# EPICS SNL sequencer program: HFMAGPSUSup/fsm_stage1.st
program fsm("P, RAMPTABLEDIR")

/* STAGE 1: This FSM can do basic ramping from point A to point B: no incremental ramping,
no direction work. */

/*
**************************************************************************
fsm.st

State Machine for the Hifi Cryomagnet PSU

- Reads ramp rate table from external file and stores targets/rates in
  two unsorted arrays: ramp_table_targets and their corresponding ramp_table_rates.

- The directory of the ramp file is passed to this script via the RAMPTABLEDIR
  macro. This is sourced from the st-common.cmd IOC file.

- Ramp file reading skips line 0, it is reserved for column headers.
  Subsequent file_liness have pairs of space-seperated values (target, rate)

- Ramping is incremental (ramps to interim points along the way) to avoid ramping too
  quickly if there is a comms error.

- the Direction PV sets the polarity of the ramp. When ramping from +ve to -ve
  (or vice-versa), we ramp to zero, flip the polarity, and continue the ramp to
  the user's target.

*************************************************************************
*/

/* INITIALISER VARIABLES */

double CONSTANT_INIT = 0.029;

#include "seqPVmacros.h"
%{#include <stdlib.h>}%
%{#include <stdio.h>}%
%{#include <float.h>}%

/* Turn on run-time debug messages */
option +d;

/* PV definitions */
PV(double, get_mid, "{P}:MID", Monitor);
PV(double, get_max, "{P}:MAX", Monitor);
PV(double, get_zero, "{P}:ZERO", Monitor);
PV(double, set_zero, "{P}:ZERO", Monitor);
PV(double, get_limit, "{P}:LIMIT", Monitor);
PV(string, get_pause, "{P}:PAUSE", Monitor);
PV(double, get_output, "{P}:OUTPUT", Monitor);
PV(double, get_constant, "{P}:CONSTANT", Monitor);
PV(double, get_ramp_rate, "{P}:RAMPRATE", Monitor);
PV(string, get_direction, "{P}:DIRECTION", Monitor);
PV(string, get_ramp_target, "{P}:RAMPTARGET", Monitor);
PV(string, get_output_mode, "{P}:OUTPUTMODE", Monitor);
PV(int, read_ramp_file_trigger, "{P}:READFILE", Monitor);
PV(string, get_heater_status, "{P}:HEATERSTATUS", Monitor);
PV(int, write_ramp_file_trigger, "{P}:WRITEFILE", Monitor);
PV(double, final_target, "{P}:MIDFINALTARGET", Monitor);

char ramp_table_directory[256]; assign ramp_table_directory to "{P}:RAMPTABLEDIRECTORY";
char temp_log[256];
double ramp_table_rates[64]; assign ramp_table_rates to "{P}:RAMPTABLERATES"; monitor ramp_table_rates;
double ramp_table_targets[64]; assign ramp_table_targets to "{P}:RAMPTABLETARGETS"; monitor ramp_table_targets;
int system_stable; assign system_stable to "{P}:SYSTEMSTABLE";

double ramp_time; assign ramp_time to "{P}:RAMPTIME"; monitor ramp_time;

double set_max; assign set_max to "{P}:MAX:SP";
double set_mid; assign set_mid to "{P}:MID:SP";
int set_pause; assign set_pause to "{P}:PAUSE:SP";
double set_limit; assign set_limit to "{P}:LIMIT:SP";
int set_ramp_target; assign set_ramp_target to "{P}:RAMPTARGET:SP";
int set_direction; assign set_direction to "{P}:DIRECTION:SP";
double set_constant; assign set_constant to "{P}:CONSTANT:SP";
double set_ramp_rate; assign set_ramp_rate to "{P}:RAMPRATE:SP";
int set_output_mode; assign set_output_mode to "{P}:OUTPUTMODE:SP";

char set_log_message[256]; assign set_log_message to "{P}:LOGMESSAGE";
int set_heater_status; assign set_heater_status to "{P}:HEATERSTATUS:SP";

/* File reading variables */
char buffer[25];
int file_lines = 0;
char *token;
char delim[2] = " ";
double sort_values[64][2];

/* Interim Ramp Rate Check Variables */

double check_difference;
int temp_target_table_index = 0;

int largest_target_index;
int smallest_target_index;

float abs_target;

int continue_ramp_after_zero_reached;
double ramp_zero_cache;
double interim_ramping_tolerance;

/* direction setters */
int POSITIVE = 2;
int NEGATIVE = 1;
/* Pause setters */
int PAUSED = 1;
int UNPAUSED = 0;
/* ramp targets */
int TARGET_ZERO = 0;
int TARGET_MID = 1;
int TARGET_MAX = 2;

/* Turn on run-time debug messages */
option +d;

%{
	/*
		Escaped C Code - this section contains functions called within states.
	*/

	static void sort_column(double arr[][2], int file_lines) {
		/*
			Function to sort ramp file values into order by target value
			This is so we can more easily find the next appropriate ramp target.
		*/
		int i,j,k;
		double key;
		for(i=0;i<file_lines;i++)
		{
			for(j=1;j<file_lines;j++)
			{
				key=arr[j][i];
				k=j-1;
				while(k>=0 && arr[k][i]>key)
				{
					arr[k+1][i]=arr[k][i];
					k--;
				}
				arr[k+1][i]=key;
			}
		}
	}

	static void read_ramp_table_rates() {
		/*
			Reading ramp table values from external .txt file
			Puts file values into ramp_table_rates and ramp_table_targets
		*/

		/* Empty our arrays for re-writing */
		memset(ramp_table_targets, -1, sizeof(ramp_table_rates));
		memset(ramp_table_rates, -1, sizeof(ramp_table_rates));
		memset(sort_values, -1, sizeof(sort_values));
		file_lines = 0;

		FILE *ramp_file;
		ramp_file = fopen(ramp_table_directory, "r");

		if (ramp_file != NULL) {
			/* Skip first line */
			fgets(buffer, 30, ramp_file);

			while (fgets(buffer, 30, ramp_file) != NULL) {
				token = strtok(buffer, delim);
				sort_values[file_lines][0] = strtod(token, NULL);
				token = strtok(NULL, delim);
				sort_values[file_lines][1] = strtod(token, NULL);
				file_lines++;
			}
		}
		else {
			printf("\nFile Read Error");
			exit(-1);
		}
		fclose(ramp_file);

		/* Sort ramp file values into ascending order of target, and put into our PV values*/
		for (int i = 0; i < file_lines;i++) {
			sort_column(sort_values, file_lines);
			ramp_table_targets[i] = sort_values[i][0];
			ramp_table_rates[i] = sort_values[i][1];
		}
	}

	static void write_ramp_table_to_file() {
		/*
			Writing ramp rate and target values to our .txt file
		*/

		printf("\n==> Writing file...");

		FILE *ramp_file;
		ramp_file = fopen(ramp_table_directory, "w");
		int j = 0;
		for(int i = 0; i < 64; i++) {
			if (ramp_table_targets[i] > 0) {
				j++;
			}
		}

		if (ramp_file != NULL) {

			fprintf(ramp_file, "target rate");

			for (int i = 0; i < j; i++) {
				if ((ramp_table_rates[i] > 0) && (ramp_table_targets[i] > 0)) {
					fprintf(ramp_file, "\n%f %f", ramp_table_targets[i], ramp_table_rates[i]);
					printf("\nWriting file_lines: %f %f", ramp_table_targets[i], ramp_table_rates[i]);
				}
			}
		}
		else {
			printf("\nFile Read Error");
			exit(-1);
		}
		fclose(ramp_file);

		printf("\n==> File write successful!");
		/* Trigger a re-read to get values in sorted order */
		read_ramp_table_rates();
	}

	static int find_nearest_ramp_rate(double current_output) {
		/*
			:returns: Index value of next available ramp target/ramp rate.

			Return of 100 indicates that we have gone beyond the ranges of the
			ramp table.
		*/

		int nearest_index = 0;
		largest_target_index = file_lines-1;
		smallest_target_index = 0;

		for (int x = 0; x < file_lines; x++) {
			/* Ramping up? Find next highest value */
			if (fabs(final_target) > fabs(current_output)) {
				if(fabs(current_output) < (ramp_table_targets[x]/10000)) {
					nearest_index = x;
					break;
				}
			}
			/* Ramping down? Find next lowest Value */
			if (fabs(final_target) < fabs(current_output)) {
				if(fabs(current_output) > (ramp_table_targets[x]/10000)) {
					nearest_index = x;
				}
			}
		}
		/* If we have reached the last table value, and our final target is beyond that - */
		if (((fabs(final_target) > (ramp_table_targets[file_lines-1]/10000)) && ( fabs(current_output) >= (ramp_table_targets[file_lines-1]/10000)) ) ||
			( ( fabs(final_target) < (ramp_table_targets[0]/10000)) && (fabs(current_output) <= (ramp_table_targets[0]/10000))) ){
			/*printf("\n==> We're heading beyond the ranges of the ramp table!");*/
			nearest_index = 100;
		}
		return nearest_index;
	}

	static double calc_ramp_duration() {
		printf("\n\n***** Calculating ramp time *******");
		double ramp_time = 0.0;
		int interim;
		int index = 0;
		double current_position = get_output*10000;
		/* ramping up? */

		if (fabs(final_target) > fabs(current_position)) {
			index = temp_target_table_index;
			while(index < file_lines) {
				if (fabs(final_target) < ramp_table_targets[index]) {
					printf("\nramp time += %f - %f * %f", final_target, current_position, (ramp_table_rates[index]*get_constant*10000));
					ramp_time += ((fabs(final_target) - current_position) * (ramp_table_rates[index]*get_constant*10000));
					index = file_lines;
				}
				else {
					ramp_time += ((ramp_table_targets[index] - current_position) * (ramp_table_rates[index]*get_constant*10000));
					printf("\nramp time += %f - %f * %f", ramp_table_targets[index], current_position, (ramp_table_rates[index]*get_constant*10000));
					printf("\nramp_time: %f \tconstant: %f", ramp_time, get_constant);
					current_position = ramp_table_targets[index];
					index += 1;
				}
			}
			/* if final target is beyond ramp table values */
			if(fabs(final_target) > ramp_table_targets[file_lines]) {
				/* if current output is currently beyond table range */
				if(current_position > ramp_table_targets[file_lines]) {
					ramp_time += ((final_target - current_position) * (ramp_table_rates[index]*get_constant*10000));
					printf("\nbeyond ramp time += %f - %f * %f", final_target, current_position, (ramp_table_rates[index]*get_constant*10000));
					printf("\nramp_time: %f", ramp_time);
				}
				else {
					ramp_time += (final_target - ramp_table_targets[file_lines] * (ramp_table_rates[file_lines]*get_constant*10000));
					printf("\n+ full beyond ramp time += %f - %f * %f", final_target, current_position, (ramp_table_rates[index]*get_constant*10000));
					printf("\nramp_time: %f", ramp_time);

				}

			}
		}
		printf("\nnew ramp time: ramp_time: %f", ramp_time);
		return ramp_time;
	}
}%

foreign ssId;

ss fsm {

	state init {

		entry {
			printf("\nhello world!");
			printf("\n==> Reading ramp table, setting limit, constant and target\n");
			strcpy(ramp_table_directory, macValueGet("RAMPTABLEDIR"));
			pvPut(ramp_table_directory, SYNC);
			read_ramp_table_rates();
			pvPut(ramp_table_rates, SYNC);
			pvPut(ramp_table_targets, SYNC);
			set_ramp_rate = ramp_table_rates[0]; pvPut(set_ramp_rate, SYNC);
			set_limit = 5.0; pvPut(set_limit, ASYNC);
			set_constant = CONSTANT_INIT; pvPut(set_constant, ASYNC);
			set_ramp_target = TARGET_MID; pvPut(set_ramp_target, SYNC);

			set_pause = PAUSED; pvPut(set_pause, SYNC);
			strcpy(set_log_message, " ==> I'm the initial log message!"); pvPut(set_log_message, SYNC);

		}

		when( fabs(get_constant-CONSTANT_INIT) < 0.01 ){
			printf("\n==> Constant set, setting outputmode, min, max\n");

		} state init2
	}

	state init2 {
		entry {
			set_output_mode = 1; pvPut(set_output_mode, SYNC);

		}
		when (strcmp(get_output_mode, "TESLA")==0) {
			printf("\n==> Output mode set, setting mid and max values");
		} state init3

	}

	state init3 {
	entry {

		set_max = 0.4; pvPut(set_max, SYNC);
		set_mid = 0.2; pvPut(set_mid, SYNC);
	}
	when (fabs(get_mid-0.4)<0.01) {
		printf("\n==> PVs all set");
	} state idle

	}

	state idle {

		entry {
			printf("\n==> idle: Waiting for system to be unpaused...");

		}

		when(strcmp(get_pause, "OFF")==0) {
			printf("\nMoving to ramping state");
		} state ramping_active

		when(write_ramp_file_trigger > 0) {
			printf("\nMoving to write_file state!");
		} state write_ramp_table_file

		when(read_ramp_file_trigger > 0) {
			printf("\nMoving to read_file state!");
		} state read_ramp_table_file

	}

	state ramping_active {

		entry {
			printf("\nramping ramping ramping");
		}
			/*strcpy(set_log_message, "RAMP STATUS: RAMPING FROM %f TO %f AT %f A/SEC", get_output*10000, get_mid, get_rate); pvPut(set_log_message, SYNC);*/
		when(strcmp(get_pause, "ON")==0) {
			printf("\npaused!");
		} state idle
	}

		state write_ramp_table_file {
		entry {
			printf("\n==> Writing ramp table file to directory...");
			write_ramp_table_to_file();
			write_ramp_file_trigger = 0; pvPut(write_ramp_file_trigger, SYNC);
		}
		when (delay(1)) {

		} state idle
	}

	state read_ramp_table_file {
		entry {
			printf("\n==> Reading ramp table file and setting PVs...");
			read_ramp_table_rates();
			pvPut(ramp_table_rates, SYNC);
			pvPut(ramp_table_targets, SYNC);
			read_ramp_file_trigger = 0; pvPut(read_ramp_file_trigger, SYNC);
		}
		when (delay(1)) {

		} state idle
	}
}
